TYPE E_RobotCommandCode : (
    ROBOT_CMD_NONE := 0,
    ROBOT_CMD_START := 10,
    ROBOT_CMD_STOP := 20,
    ROBOT_CMD_INITIALIZE := 30,
    ROBOT_CMD_RESET := 40,
    ROBOT_CMD_ABORT := 50
); END_TYPE

(* stored: Version 1.1.0.1
   DUT E_RobotCommandCode: Id {E3000000-0000-4000-8000-000000000024} *)
